{attribute 'enable_dynamic_creation'}
{attribute 'no_explicit_call' := 'do not call this FB directly'}
FUNCTION_BLOCK PUBLIC DirectoryEntry EXTENDS FileSystemEntry IMPLEMENTS I_DirectoryEntry
VAR
END_VAR

PROPERTY PUBLIC IsDirectory : BOOL
GET
IsDirectory := TRUE;
END_GET
END_PROPERTY

END_FUNCTION_BLOCK

(* stored: Version 1.1.0.1, ProductVersion 3.1.4024.9
   POU DirectoryEntry: Id {41f8ec17-6d67-40fc-801c-f71f51d87d59}, SpecialFunc None
   Property IsDirectory: Id {8bc2465d-80f6-4f35-99d3-38286b545c90}
   Get Get: Id {6ed72c3e-b222-4fef-830b-c3836eee6ac4} *)
